{attribute 'GeneratedUsingTerminal: EL2912-0000-0016'}
{attribute addProperty BoxType "EL2912-0000-0016"}
{attribute addProperty Id "EtcSlaveTerminalBaseModule_1_FSOEModule_1_FSOE_263516AE16Module_2_FSOUTModule_2_FSOUT_6D5CB05D2Module_3_DEVICEIOModule_3_DEVICEIO_5FA6B4E72Module_4_FSLOGICModule_4_FSLOGIC_DEAB45222WcStateAT %I*WcState_B516A2644InfoDataAT %I*InfoData_32EB74EA10"}
{attribute addProperty CRC "3465745356"}
{attribute addProperty Size "36"}
TYPE EL2912_CE9313CC EXTENDS EtcSlaveTerminalBase :
STRUCT
	{attribute addProperty Name "Module_1_FSOE"}
	Module_1_FSOE : Module_1_FSOE_263516AE;
	{attribute addProperty Name "Module_2_FSOUT"}
	Module_2_FSOUT : Module_2_FSOUT_6D5CB05D;
	{attribute addProperty Name "Module_3_DEVICEIO"}
	Module_3_DEVICEIO : Module_3_DEVICEIO_5FA6B4E7;
	{attribute addProperty Name "Module_4_FSLOGIC"}
	Module_4_FSLOGIC : Module_4_FSLOGIC_DEAB4522;
	{attribute addProperty Name "WcState"}
	WcState : WcState_B516A264;
	{attribute addProperty Name "InfoData"}
	InfoData : InfoData_32EB74EA;
END_STRUCT
END_TYPE

(* stored: Version 1.2.0.0, ProductVersion 3.1.4024.9
   DUT EL2912_CE9313CC: Id {0228644b-fa91-49b4-9c7b-4d963f629553} *)
